(* CODESYS project cylinders_initial_RECOVERED_2023-08-31T10-13-54.project

Project tree, tasks and I/O mapping:
  Device : CODESYS Control Win V3, 3S - Smart Software Solutions GmbH, version 3.5.16.0
    application Application
      libraries: Standard, * (System); CmpBitmapPool, * (System); Util, * (System)
      task MainTask (cyclic, interval 5 ms, priority 1) calls cylinder_ctrl
      task simulation (cyclic, interval t#20ms, priority 1) calls sim_logic
      task VISU_TASK (cyclic, interval 10 ms, priority 31) calls VisuElems.Visu_Prg
      visualisation Cylinders
      global variables IO
      control/
        program cylinder_ctrl [LD]
      simulation/
        program sim_logic [LD]
        function block cylSimulation [ST]
      image pool ImagePool
  libraries: VisuSymbols, 3.5.10.0 (System)
  5ce3da45-db07-42e7-a21c-a00fff4ed8f6|C:\Users\ryytt\OneDrive\Skrivbord\examensarbete\bakgrund.png
  5ce3da45-db07-42e7-a21c-a00fff4ed8f6|C:\Users\ryytt\OneDrive\Skrivbord\examensarbete\bakgrundv2.png
  text list GlobalTextList
*)

// Device/Application/IO
VAR_GLOBAL
	ixStart: BOOL; // the start switch and the button
 	ixStop: BOOL;  // the stop switch and the button
	ixReset: BOOL; // the reset switch
	ixB1: BOOL; // button B1
	ixB2: BOOL; // button B2
	ixIN10: BOOL; // the IN10 switch
	ixIN11: BOOL; // the IN11 switch
	ixCylinder1In: BOOL; // a sensor if cylinder 1 is in
	ixCylinder1Out: BOOL; // a sensor if cylinder 1 is in
	ixCylinder2In: BOOL; // a sensor if cylinder 1 is in
	ixCylinder2Out: BOOL; // a sensor if cylinder 1 is in
	ixCylinder3In: BOOL; // a sensor if cylinder 1 is in
	ixCylinder3Out: BOOL; // a sensor if cylinder 1 is in	
	ixEmergencyStop: BOOL := TRUE; // the emergency stop. If false, it is active

	qxLamp1: BOOL; // to control L1
	qxLamp2: BOOL; // to control L2
	qxLamp3: BOOL; // to ontorl L3
	qxLamp4: BOOL; // to control L4
	qxCylinder1: BOOL; // to extend cylinder 1
	qxCylinder2: BOOL; // to extend cylinder 2
	qxCylinder3: BOOL; // to extend cylinder 3
END_VAR

// Device/Application/control/cylinder_ctrl
PROGRAM cylinder_ctrl
VAR
END_VAR

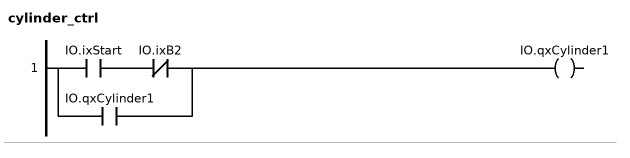
// NETWORK 1
IO.qxCylinder1 := IO.ixStart AND NOT IO.ixB2 OR IO.qxCylinder1;

END_PROGRAM

// Device/Application/simulation/sim_logic
PROGRAM sim_logic
VAR
	cyl1: cylSimulation;
	donotuse_cyl1_pos: INT;
	cyl2: cylSimulation;
	cyl3: cylSimulation;
	donotuse_cyl2_pos: INT;
	donotuse_cyl3_pos: INT;
END_VAR

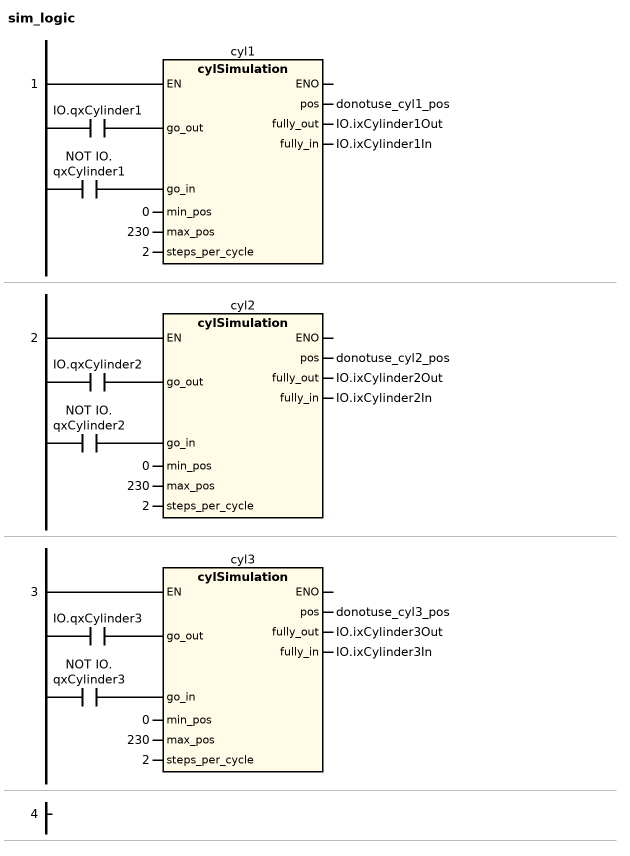
// NETWORK 1
cyl1(
    go_out := IO.qxCylinder1,
    go_in := NOT IO.qxCylinder1,
    min_pos := 0,
    max_pos := 230,
    steps_per_cycle := 2,
    pos => donotuse_cyl1_pos,
    fully_out => IO.ixCylinder1Out,
    fully_in => IO.ixCylinder1In); // cylSimulation

// NETWORK 2
cyl2(
    go_out := IO.qxCylinder2,
    go_in := NOT IO.qxCylinder2,
    min_pos := 0,
    max_pos := 230,
    steps_per_cycle := 2,
    pos => donotuse_cyl2_pos,
    fully_out => IO.ixCylinder2Out,
    fully_in => IO.ixCylinder2In); // cylSimulation

// NETWORK 3
cyl3(
    go_out := IO.qxCylinder3,
    go_in := NOT IO.qxCylinder3,
    min_pos := 0,
    max_pos := 230,
    steps_per_cycle := 2,
    pos => donotuse_cyl3_pos,
    fully_out => IO.ixCylinder3Out,
    fully_in => IO.ixCylinder3In); // cylSimulation

// NETWORK 4

END_PROGRAM

// Device/Application/simulation/cylSimulation
FUNCTION_BLOCK cylSimulation
VAR_INPUT
	go_out: BOOL;
	go_in: BOOL;
	min_pos: INT;
	max_pos: INT;
	steps_per_cycle: INT;
END_VAR
VAR_OUTPUT
	pos: INT;
	fully_out: BOOL;
	fully_in: BOOL;
END_VAR
VAR
END_VAR


IF go_out AND NOT go_in THEN
	pos := pos + steps_per_cycle;
END_IF
IF go_in AND NOT go_out THEN
	pos := pos - steps_per_cycle;
END_IF

pos := LIMIT(min_pos, pos, max_pos);

fully_in := pos = min_pos;
fully_out := pos = max_pos;

END_FUNCTION_BLOCK

// Device/Application/Cylinders
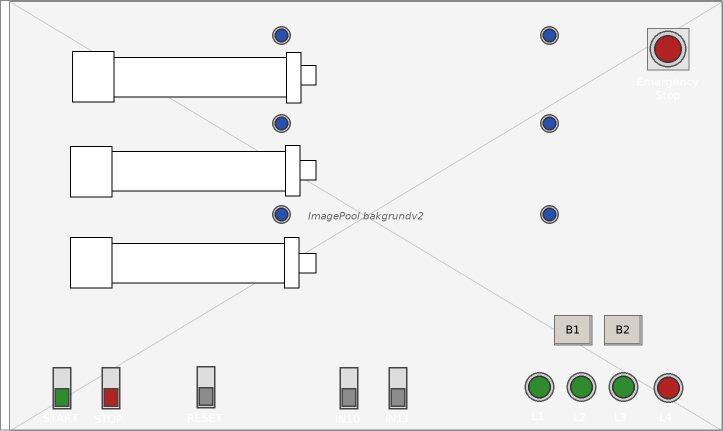
VISUALIZATION Cylinders  // 723x431
    Image (9,1 714x430), image: ImagePool.bakgrundv2
    Rectangle (286,253 30x20)
        p874137650: sim_logic.donotuse_cyl3_pos
    Rectangle (286,160 30x20)
        p874137650: sim_logic.donotuse_cyl2_pos
    Lamp1 (522,370 35x34), tooltip "L1", variable: qxLamp1, style: Lamp-Lamp1-Green
    Lamp1 (564,370 35x34), tooltip "L2", variable: qxLamp2, style: Lamp-Lamp1-Green
    Lamp1 (606,370 35x34), tooltip "L3", variable: qxLamp3, style: Lamp-Lamp1-Green
    Lamp1 (651,371 35x34), tooltip "L4", variable: qxLamp4, style: Lamp-Lamp1-Red
    DipSwitch (41,366 42x44), variable: ixStart, behaviour: TOGGLE, style: Switch-DipSwitch-Green
    DipSwitch (90,366 42x44), variable: ixStop, behaviour: TOGGLE, style: Switch-DipSwitch-Red
    DipSwitch (185,365 42x44), tooltip "RESET", variable: ixReset, behaviour: TOGGLE, style: Switch-DipSwitch-Gray
    DipSwitch (328,366 42x44), variable: ixIN10, behaviour: TOGGLE, style: Switch-DipSwitch-Gray
    DipSwitch (377,366 42x44), variable: ixIN11, behaviour: TOGGLE, style: Switch-DipSwitch-Gray
    Label (16,409 89x19), "START"
    Label (64,410 89x19), "STOP"
    Label (160,409 89x19), "RESET"
    Label (303,410 89x19), "IN10"
    Label (353,409 89x19), "IN11"
    Label (493,407 89x19), "L1"
    Label (535,408 89x19), "L2"
    Label (576,408 89x19), "L3"
    Label (621,408 89x19), "L4"
    Rectangle (286,65 30x20)
        p874137650: sim_logic.donotuse_cyl1_pos
    Rectangle (101,57 193x40)
    Rectangle (99,151 193x40)
    Rectangle (102,243 193x40)
    RoundedRectangle (70,237 42x51), "CYL3"
    RoundedRectangle (70,146 42x51), "CYL2"
    RoundedRectangle (72,51 42x51), "CYL1"
    RoundedRectangle (286,52 15x51)
    RoundedRectangle (285,145 15x51)
    RoundedRectangle (284,237 15x51)
    Lamp1 (271,25 21x21), variable: ixCylinder1In, style: Lamp-Lamp1-Blue
    Lamp1 (539,25 21x21), variable: ixCylinder1Out, style: Lamp-Lamp1-Blue
    Lamp1 (271,113 21x21), variable: ixCylinder2In, style: Lamp-Lamp1-Blue
    Lamp1 (539,113 21x21), variable: ixCylinder2Out, style: Lamp-Lamp1-Blue
    Lamp1 (271,204 21x21), variable: ixCylinder3In, style: Lamp-Lamp1-Blue
    Lamp1 (539,204 21x21), variable: ixCylinder3Out, style: Lamp-Lamp1-Blue
    PushSwitch (647,27 42x44), variable: ixEmergencyStop, behaviour: TOGGLE, style: Switch-PushSwitch-Red
    Label (623,72 90x33), "Emergency Stop"
    Button (554,315 38x30), "B1"
        tap ixB1
    Button (604,315 38x30), "B2"
        tap ixB2
END_VISUALIZATION
